% RSLogix 500 project SARAN G 181EI154_BAK039.RSS, saved by version 8.10.00.18 %
PROJECT "UNTITLED"    % processor: MicroLogix 1200 %

PROGRAM FILES
  LAD 2   11 rungs

DATA FILES
  O0 OUTPUT  4 elements
  I1 INPUT  4 elements
  S2 STATUS  66 elements
  B3 BINARY  1 elements
  T4 TIMER  4 elements
  C5 COUNTER  1 elements
  R6 CONTROL  1 elements
  N7 INTEGER  1 elements

LADDER 2
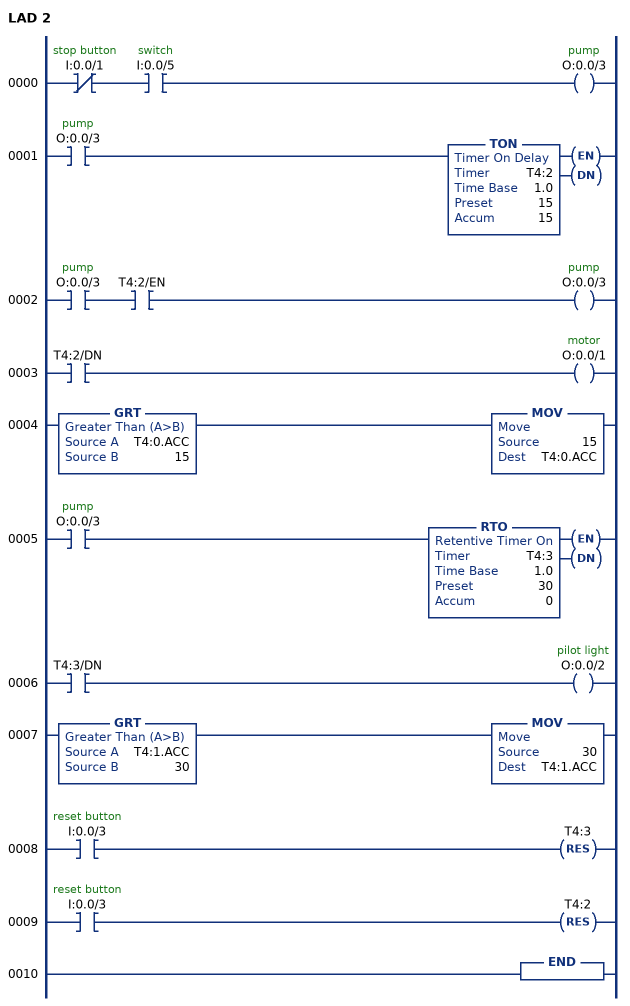
% Rung: 0 %
SOR XIO I:0.0/1 XIC I:0.0/5 OTE O:0.0/3 EOR
%   I:0.0/1  "stop button" %
%   I:0.0/5  "switch" %
%   O:0.0/3  "pump" %
% Rung: 1 %
SOR XIC O:0.0/3 TON T4:2 1.0 15 15 EOR
%   O:0.0/3  "pump" %
% Rung: 2 %
SOR XIC O:0.0/3 XIC T4:2/EN OTE O:0.0/3 EOR
%   O:0.0/3  "pump" %
% Rung: 3 %
SOR XIC T4:2/DN OTE O:0.0/1 EOR
%   O:0.0/1  "motor" %
% Rung: 4 %
SOR GRT T4:0.ACC 15 MOV 15 T4:0.ACC EOR
% Rung: 5 %
SOR XIC O:0.0/3 RTO T4:3 1.0 30 0 EOR
%   O:0.0/3  "pump" %
% Rung: 6 %
SOR XIC T4:3/DN OTE O:0.0/2 EOR
%   O:0.0/2  "pilot light" %
% Rung: 7 %
SOR GRT T4:1.ACC 30 MOV 30 T4:1.ACC EOR
% Rung: 8 %
SOR XIC I:0.0/3 RES T4:3 EOR
%   I:0.0/3  "reset button" %
% Rung: 9 %
SOR XIC I:0.0/3 RES T4:2 EOR
%   I:0.0/3  "reset button" %
% Rung: 10 %
SOR END EOR

OTHER DOCUMENTED ADDRESSES
  I:0.0/0  "switch"
  O:0.0/0  "pump"

DATA TABLE (non-zero values as saved)
DATA T4
% .PRE .ACC %
% T4:0 % 15 15
% T4:1 % 30 0
% T4:2 % 15 15
% T4:3 % 30 0
